{attribute 'GeneratedUsingTerminal: CU1124-0000-0016'}
{attribute addProperty BoxType "CU1124-0000-0016"}
{attribute addProperty Id "A_0004_CU1128_0000_0000A_0004_CU1128_0000_0000_C48505B892"}
{attribute addProperty CRC "1949799616"}
{attribute addProperty Size "92"}
TYPE A_0003_CU1124_0000_0016_743794C0 EXTENDS CU1124_1FC0878B :
STRUCT
	{attribute addProperty Name "A_0004_CU1128_0000_0000"}
	{attribute addProperty PreviousPort "A_0003(CU1124-0000-0016) : D"}
	A_0004_CU1128_0000_0000 : A_0004_CU1128_0000_0000_C48505B8;
END_STRUCT
END_TYPE

(* stored: Version 1.2.0.0, ProductVersion 3.1.4024.9
   DUT A_0003_CU1124_0000_0016_743794C0: Id {eac46921-ff77-470f-9011-c7110cbe0a5e} *)
